INTERFACE I_SimpleLogPublisher EXTENDS I_Base

METHOD Subscribe
VAR_INPUT
	Logger : I_SimpleLogger;
END_VAR
END_METHOD

END_INTERFACE

(* stored: Version 1.1.0.1
   Itf I_SimpleLogPublisher: Id {637a1c51-6794-4701-a99d-e58d0530dad3}
   Method Subscribe: Id {204c1bed-d99d-4512-a1d0-63490e307fb1} *)
